(* CoDeSys 2.3 project: log-lib-all.pro *)
(* Libraries: Standard.lib 20.3.12 18:22:36, Smi_plc.lib 20.3.12 18:22:36 *)

(* PLC configuration (modules and I/O channels)
I/O modules [BE_IO_MODULE_FOLDER] node 1, in %IB0 out %QB0 {WordType = 256}
CAN-Netze [BE_CAN_NETWORKS_FOLDER] node 2, in %IB0 out %QB0 {WordType = 256}
ProfiBus-Netze [BE_PB_NETWORKS_FOLDER] node 3, in %IB0 out %QB0 {WordType = 256}
Networks [BE_NETWORKS_FOLDER] node 4, in %IB0 out %QB0 {WordType = 256}
*)

(* POU PLC_PRG, ST *)
PROGRAM PLC_PRG
VAR
END_VAR
(*
 * README
 * 
 * 
 *)
;
END_PROGRAM
